INTERFACE I_Link

// Get/set if the link needs to be excluded from the links overview
PROPERTY ExcludeFromOverview : BOOL
GET
END_GET
SET
END_SET
END_PROPERTY

// Group of inputs
PROPERTY InputGroup : I_DIGroup
GET
END_GET
SET
END_SET
END_PROPERTY

// Group of outputs
PROPERTY OutputGroup : I_DOGroup
GET
END_GET
SET
END_SET
END_PROPERTY

// Output reaction
PROPERTY OutputReaction : REFERENCE TO ST_CommandTranslation
GET
END_GET
END_PROPERTY

END_INTERFACE

(* stored: Version 1.1.0.1, ProductVersion 3.1.4024.12
   Itf I_Link: Id {04cab8aa-8b6c-4150-a2fd-0c4775e771ff}
   Folder Properties: Id {d3758d61-f435-4656-9eff-9b20d008ef4a}
   Property ExcludeFromOverview: Id {e7a80a3a-f2eb-4939-b1f8-9f0a5fff8c15}
   Get Get: Id {9ea60335-bb8f-414c-b646-f5c0e2209c90}
   Set Set: Id {7dc2ad2b-c4a2-424f-addb-29b887e14e0d}
   Property InputGroup: Id {8a3382ce-fc11-432e-b0be-1163f5a1d7ee}
   Get Get: Id {8c768c7c-3031-429b-acd5-3c405fa88487}
   Set Set: Id {94833dc0-77e7-40bc-9b7a-04607a5883f8}
   Property OutputGroup: Id {1036a780-dec2-42ee-9f72-df6d5c79c06b}
   Get Get: Id {1236f278-ff8b-4a03-8076-aea1611c0b7b}
   Set Set: Id {13a04904-07f8-4e68-bbd1-3b22a38309d8}
   Property OutputReaction: Id {d1db3345-c9f3-408c-8b05-4b08ab7283b3}
   Get Get: Id {cf5961d1-69ce-4359-af40-0c4037411f05} *)
